// Mitsubishi GX Works2 project: PLC_Mitsubishi   PLC: Q04UDEH

PROGRAM MAIN
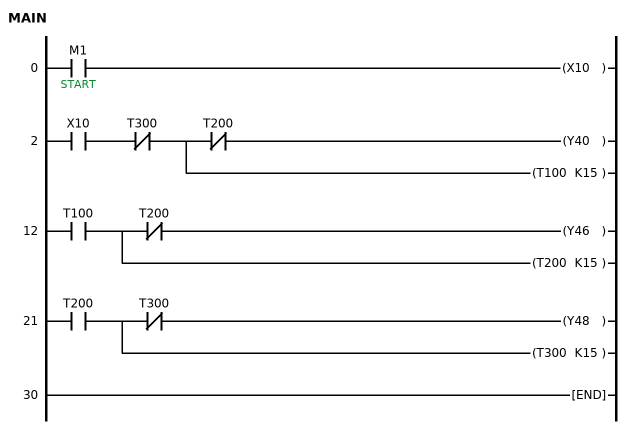
0     LD      M1  ; START
      OUT     X10
2     LD      X10
      ANI     T300
      MPS
      ANI     T200
      OUT     Y40
      MPP
      OUT     T100 K15
12    LD      T100
      MPS
      ANI     T200
      OUT     Y46
      MPP
      OUT     T200 K15
21    LD      T200
      MPS
      ANI     T300
      OUT     Y48
      MPP
      OUT     T300 K15
30    END
END_PROGRAM

// device comments not shown above
M2  ; STOP
